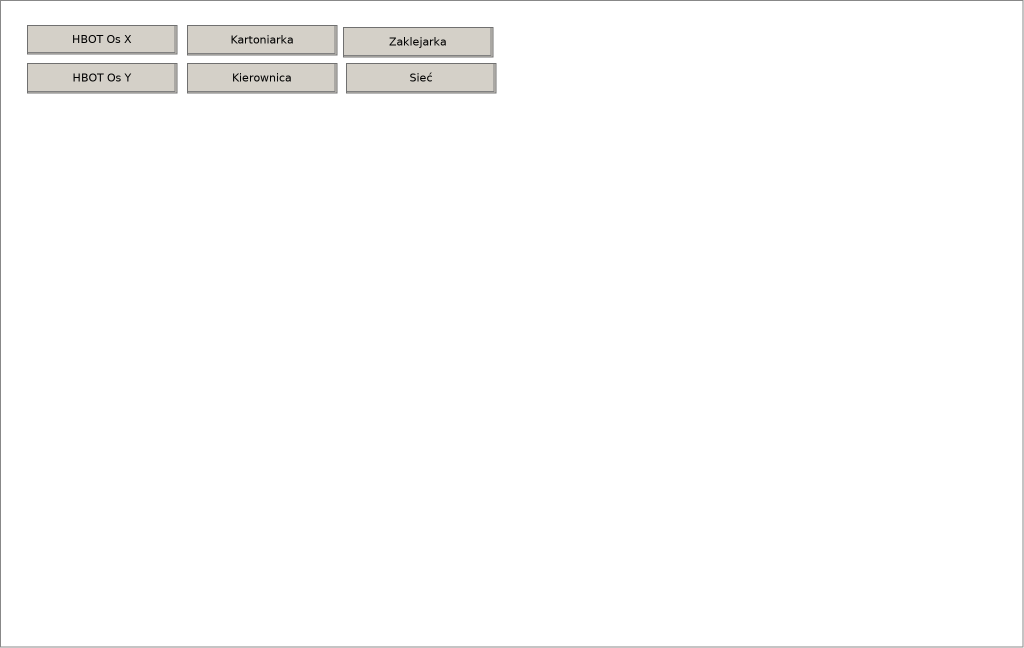
VISUALIZATION Serwis  // 1024x648
    Button (27,25 150x29), "HBOT Os X", colour toggle: GVL_HMI.strona_1=2
        OnMouseDown: FrameSelectionChange Selection=SelectedFrame=9731c5c5-429f-486e-9358-6f2f3bdb5ae0, GlobSel=AssignType=Directly, SelType=Locally
        OnMouseDown: execute { GVL_HMI.strona_1:=2; }
    Button (187,25 150x30), "Kartoniarka"
    Button (343,27 150x30), "Zaklejarka"
    Button (187,63 150x30), "Kierownica"
    Button (346,63 150x30), "Sieć"
    Button (27,63 150x30), "HBOT Os Y", colour toggle: GVL_HMI.strona_1=1
        OnMouseDown: FrameSelectionChange Selection=SelectedFrame=9731c5c5-429f-486e-9358-6f2f3bdb5ae0, Selection=1, GlobSel=AssignType=Directly, SelType=Locally
        OnMouseDown: execute { GVL_HMI.strona_1:=1; }
END_VISUALIZATION

(* stored: Version 1.1.0.1, ProductVersion 3.1.4022.12
   Visu Serwis: Id {067415b4-5022-450f-83c9-14559d8141cf} *)
